# B&R Automation Studio project lihui1
Automation Studio 4.6.3.55 SP

## Configuration Config1

CPU X20CP1586, AutomationRuntime B4.63, Build 4.1.2, Vc V4.62.0

### Task classes (Cpu.sw)
```
Cyclic#4:
  Program <- Program.prg
Cyclic#7:
  RevInfo <- RevInfo.RevInfo.prg
Libraries: AsBrStr
```

### Hardware
```
X20CP1586 : X20CP1586 v1.5.0.0
  Connector IF2:
    ActivateDevice = 1
  ConfigurationID = lihui1_Config1
  Simulation = 1
```

## Logical view

### Program Logical/Program (IEC)

#### Init.ab - Init code
```automation-basic
PROGRAM _INIT
	(* Insert code here *)

END_PROGRAM
```

#### Exit.ab - Exit code
```automation-basic
PROGRAM _EXIT
	(* Insert code here *)

END_PROGRAM
```

#### Variables.var - Local variables
```iecst
VAR
	PLC : USINT;
END_VAR
```

Listed in the project but not available here: Logical/Global.typ, Logical/Global.var, Logical/Libraries, Logical/RevInfo/RevInfo.var, Logical/RevInfo/RevInfo, Logical/Program/Cyclic.ab, Logical/Program/Types.typ
